Universal Robots PolyScope program: Davis_Camera_Demo_2.urp

Program Davis_Camera_Demo_2 (installation=default directory=/programs createdIn=5.20.0 lastSavedIn=5.20.0 robotSerialNumber=20245501140)
Calibrated DH parameters: a=[0.000167, -0.150231, -0.362642, 0.00007, 0.000048, 0]; d=[0.162529, 208.241507, -177.946331, -30.161797, 0.099788, 0.099549]; alpha=[1.569698, 0.001912, 0.004952, 1.572466, -1.57064, 0]; deltaTheta=[0, 1.210022, -0.817813, -0.392217, -0.000001, 0]
InitVariablesNode variables(variable(name=EyesPickAppr, expression=p[0.0,0.0,0.0,0.0,0.0,0.0]), variable(name=EyesPickPose, expression=p[0.0,0.0,0.0,0.0,0.0,0.0]), variable(name=EyesWorkpCoun_2, expression=-1), variable(name=EyesWorkpPose_2, expression=p[0.0,0.0,0.0,0.0,0.0,0.0]), variable(name=EyesWorkpiece_2, expression=-1))
Robot Program (runOnlyOnce=false)
  Loop Forever
    URCap RG Grip (OnRobot, OnRobot A/S) dataModel(rg-target-force=40.0, rg-target-width=0.1)
    MoveJ speed 60 deg/s, acceleration 80 deg/s^2 (useActiveTCP=true) feature=Base
      SuppressedNode
        Waypoint H: TCP in base x=502.604 y=-53.469 z=415.584 mm, rx=-2.349 ry=2.0268 rz=-0.0101 rad; joints [8.548, -92.361, -64.563, 248.852, -268.659, 0.001] deg; TCP offset x=0 y=0 z=230.5 mm, rx=0 ry=0 rz=0 rad
      Waypoint Home_Pose: TCP in base x=504.981 y=-52.751 z=446.833 mm, rx=-2.2448 ry=2.0973 rz=-0.042 rad; joints [8.549, -92.827, -59.612, 246.51, -268.601, 4.546] deg; TCP offset x=0 y=0 z=231.2 mm, rx=0 ry=0 rz=0 rad
      SuppressedNode
        URCap Eyes Locate (OnRobot, OnRobot A/S) dataModel(eye-process-uid=2, eye-program-calib=0)
          URCap Eyes Get Workpiece (OnRobot, OnRobot A/S) dataModel(programTypeKey=0, programCalibTypeKey=0, countAssignmentKey=EyesWorkpCount≔eyes_workp_cnt, locatePoseAssignmentKey=EyesWorkpPose≔eyes_workp_pose, workpieceAssignmentKey=EyesWorkpiece≔eyes_workp_type, Variable(key=objCntKey, variable(name=EyesWorkpCount, initializeExpression=-1)), Variable(key=objPosKey, variable(name=EyesWorkpPose, initializeExpression=p[0.0,0.0,0.0,0.0,0.0,0.0])), Variable(key=objResKey, variable(name=EyesWorkpiece, initializeExpression=-1))); state(isChildrenLocked=true)
            EyesWorkpCount := eyes_workp_cnt
            EyesWorkpPose := eyes_workp_pose
            EyesWorkpiece := eyes_workp_type
            Folder Commands
              URCap Eyes Get Workpiece (OnRobot, OnRobot A/S) dataModel(programTypeKey=0, programCalibTypeKey=0, countAssignmentKey=EyesWorkpCoun_1≔eyes_workp_cnt, locatePoseAssignmentKey=EyesWorkpPose_1≔eyes_workp_pose, workpieceAssignmentKey=EyesWorkpiece_1≔eyes_workp_type, Variable(key=objCntKey, variable(name=EyesWorkpCoun_1, initializeExpression=-1)), Variable(key=objPosKey, variable(name=EyesWorkpPose_1, initializeExpression=p[0.0,0.0,0.0,0.0,0.0,0.0])), Variable(key=objResKey, variable(name=EyesWorkpiece_1, initializeExpression=-1))); state(isChildrenLocked=true)
                EyesWorkpCoun_1 := eyes_workp_cnt
                EyesWorkpPose_1 := eyes_workp_pose
                EyesWorkpiece_1 := eyes_workp_type
                Folder Command
                  Placeholder
      URCap Eyes Locate (OnRobot, OnRobot A/S) dataModel(eye-process-uid=5, eye-program-calib=0)
        URCap Eyes Get Workpiece (OnRobot, OnRobot A/S) dataModel(programTypeKey=0, programCalibTypeKey=0, countAssignmentKey=EyesWorkpCoun_2≔eyes_workp_cnt, locatePoseAssignmentKey=EyesWorkpPose_2≔eyes_workp_pose, workpieceAssignmentKey=EyesWorkpiece_2≔eyes_workp_type, workpieceTypeKey=1, Variable(key=objCntKey, variable(name=EyesWorkpCoun_2, initializeExpression=-1)), Variable(key=objPosKey, variable(name=EyesWorkpPose_2, initializeExpression=p[0.0,0.0,0.0,0.0,0.0,0.0])), Variable(key=objResKey, variable(name=EyesWorkpiece_2, initializeExpression=-1))); state(isChildrenLocked=true)
          EyesWorkpCoun_2 := eyes_workp_cnt
          EyesWorkpPose_2 := eyes_workp_pose
          EyesWorkpiece_2 := eyes_workp_type
          Folder Commands
            URCap Eyes Pick (OnRobot, OnRobot A/S) dataModel(Variable(key=eyePickApproachPoseKey, variable(name=EyesPickAppr, initializeExpression=p[0.0,0.0,0.0,0.0,0.0,0.0])), Variable(key=eyePickPoseKey, variable(name=EyesPickPose, initializeExpression=p[0.0,0.0,0.0,0.0,0.0,0.0]))); state(isChildrenLocked=true)
              URCap TCP (OnRobot, OnRobot A/S) dataModel(tool-index=1)
              MoveJ speed 60 deg/s, acceleration 80 deg/s^2 (useActiveTCP=false) tcp=OnRobot_Default; feature=Base
                Waypoint Variable (Variable): variable=EyesPickAppr
              MoveL speed 250 mm/s, acceleration 1200 mm/s^2 (useActiveTCP=false) tcp=OnRobot_Default; feature=Base
                Waypoint Variable (Variable): variable=EyesPickPose
              URCap RG Grip (OnRobot, OnRobot A/S) dataModel(tool-index=1, rg-target-force=40.0, Variable(key=on_return, variable(name=on_return)))
              MoveL speed 250 mm/s, acceleration 1200 mm/s^2 (useActiveTCP=false) tcp=OnRobot_Default; feature=Base
                Waypoint Variable (Variable): variable=EyesPickAppr
  URCap RG Grip (OnRobot, OnRobot A/S) dataModel(rg-target-force=40.0)
